// TwinCAT 3 PLC project MainControl
// ProgramVersion: 3.1.4023.0
// libraries:
//   Tc2_Standard, * (Beckhoff Automation GmbH)
//   Tc2_System, * (Beckhoff Automation GmbH)
//   Tc3_Module, * (Beckhoff Automation GmbH)
// project tree:
//   / PlcTask.TcTTO
//   POUs/ MAIN.TcPOU
// real-time tasks:
//   TASK PlcTask: cycle T#10ms, priority 20, ADS port 350
// I/O:
//   DEVICE Gerät 4 (EtherCAT Slave), AmsNetId 5.93.125.76.5.255
//   DEVICE Gerät 1 (EtherCAT), AmsNetId 5.93.125.76.2.1
//     Klemme 1 (EK1100) [EK1100 EtherCAT-Koppler (2A E-Bus)]
//       Klemme 2 (EL6001) [EL6001 Schnittstelle (RS232)]
//       Klemme 3 (EL9011) [EL9011 Endklemme]
// variable links:
//   MainControl/MainControl Instance <-> Device 1 (EtherCAT)/Term 1 (EK1100)/Term 2 (EL6001)
//     PlcTask Inputs/MAIN.iKlemme <-> COM Inputs/Data In 0
//   MainControl/MainControl Instance <-> Device 4 (EtherCAT Slave)
//     PlcTask Inputs/MAIN.iTest <-> Inputs/Var 1
//     PlcTask Outputs/MAIN.iOut <-> Outputs/Var 91

CONFIGURATION MainControl
    RESOURCE PLC ON TwinCAT3
        TASK PlcTask(INTERVAL := T#10ms, PRIORITY := 20);
        PROGRAM MAIN WITH PlcTask : MAIN;
    END_RESOURCE
END_CONFIGURATION

// ---- POUs/MAIN.TcPOU
PROGRAM MAIN
VAR
	iTest AT %I* : INT;
	iTest2 : INT := 0;
	
	iKlemme AT %I* : USINT;
	iOut AT %Q* : USINT;
END_VAR

iTest2 := iKlemme;

iOut := iKlemme;

END_PROGRAM
